PROGRAM ClearRecipe
VAR
	i: INT;
	j: INT;
END_VAR

//Manual Logic for Reactors.Valves
	
FOR i:=0 TO 1 DO
	FOR j :=0 TO 7 DO
		IO.Reactors[i].Valves[j].bStart :=	FALSE;
	END_FOR
END_FOR
	
	//Manual Logic for Reactors.Pumps
	
FOR i:=0 TO 1 DO
	FOR j :=0 TO 1 DO
		IO.Reactors[i].Pumps[j].bStart :=FALSE;
	END_FOR
END_FOR

FOR i := 0 TO 699 DO
	RecipeTags.Recipe.Blocks[i].Properties.bBlockStarted := FALSE;
	RecipeTags.Recipe.Blocks[i].Properties.bStartCommand := FALSE;
	RecipeTags.Recipe.Blocks[i].Properties.bBlockEnded := FALSE;
	RecipeTags.Recipe.Blocks[i].Properties.bStopCommand := FALSE;
	RecipeTags.Recipe.Blocks[i].Properties.bModeSelection := FALSE;
	RecipeTags.Recipe.Blocks[i].Properties.sStartTime := '';
	RecipeTags.Recipe.Blocks[i].Properties.sEndTime := '';
	
	RecipeTags.SlaveRecipe.Blocks[i].Properties.bBlockStarted := FALSE;
	RecipeTags.SlaveRecipe.Blocks[i].Properties.bStartCommand := FALSE;
	RecipeTags.SlaveRecipe.Blocks[i].Properties.bBlockEnded := FALSE;
	RecipeTags.SlaveRecipe.Blocks[i].Properties.bStopCommand := FALSE;
	RecipeTags.SlaveRecipe.Blocks[i].Properties.bModeSelection := FALSE;
	RecipeTags.SlaveRecipe.Blocks[i].Properties.sStartTime := '';
	RecipeTags.SlaveRecipe.Blocks[i].Properties.sEndTime := '';
	
	RecipeTags.bBlockStart[i] := FALSE;
	RecipeTags.enWaitPause[i] := FALSE;
	RecipeTags.bBlockEnd[i] := FALSE;
	RecipeTags.bStartTimeEnable[i] := FALSE;

END_FOR


FOR i := 0 TO 2 DO
	IO.Reactors[i].VFD.bStart := FALSE;
	IO.Reactors[i].VFD.nRPMSetPointScaled := 0; 
END_FOR

FOR i:=0 TO 8 DO
	FOR j :=0 TO 7 DO
		IO.Vessels[i].Valves[j].bStart := FALSE;
	END_FOR
END_FOR
	
	//Manual Logic for Vessels.Pumps
	
FOR i:=0 TO 8 DO
	FOR j :=0 TO 1 DO
		IO.Vessels[i].Pumps[j].bStart :=FALSE;
	END_FOR
END_FOR

RecipeTags.bDrainStatus := FALSE;
RecipeTags.bSkipDrain := FALSE;
RecipeTags.bPauseRecipe := FALSE;
RecipeTags.bTransferStartTime	 := FALSE;

END_PROGRAM

(* stored: Version 1.1.0.1, ProductVersion 3.1.4024.5
   POU ClearRecipe: Id {a54f7d6b-5f74-425e-a1dd-d3a56698d305}, SpecialFunc None *)
